KUKA KRL program: wkz1_ab.src, wkz1_ab.dat

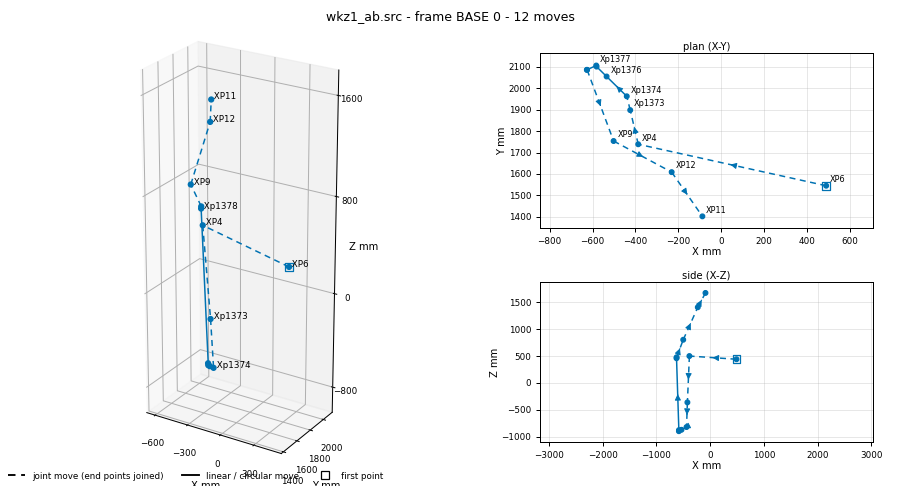
[picture p0: tool path of wkz1_ab.src in frame BASE 0, 12 of 12 moves have a stored position in this frame; points joined in program order, loops and branches not executed]
--- wkz1_ab.src ---
&ACCESS RVP6
&REL 69
&COMMENT Deposita GUN C1
DEF wkz1_ab( )
  ;FOLD INI;%{PE}%V2.2.2,%MKUKATPBASIS,%CINIT,%VCOMMON,%P
  ;FOLD BAS INI;%{PE}%V2.2.2,%MKUKATPBASIS,%CINIT,%VINIT,%P
  INTERRUPT DECL 3 WHEN $STOPMESS==TRUE DO IR_STOPM ( )
  INTERRUPT ON 3
  BAS (#INITMOV,0 )
  ;ENDFOLD
  ;FOLD A20 INI;%{E}%V2.2.2,%MKUKATPA20,%CINIT,%VINIT,%P
  IF ARC20==TRUE THEN
    A20 (ARC_INI)
    INTERRUPT DECL 6 WHEN $CYCFLAG[3]==FALSE DO A20(TECH_STOP2)
  ENDIF
  ;ENDFOLD
  ;FOLD A10 INI;%{E}%V2.2.2,%MKUKATPARC,%CINIT,%VINIT,%P
  IF A10_OPTION==#ACTIVE THEN
    INTERRUPT DECL 4 WHEN $CYCFLAG[2]==FALSE DO A10 (#APPL_ERROR)
    INTERRUPT DECL 7 WHEN A_ARC_SWI==#ACTIVE DO A10 (#ARC_SEAM)
    INTERRUPT DECL 5 WHEN A_FLY_ARC==TRUE DO A10 (#HPU_ARC)
    INTERRUPT  ON 5
    A10_INI ( )
  ENDIF
  ;ENDFOLD
  ;FOLD GRIPPER INI;%{E}%V2.2.2,%MKUKATPGRIPPER,%CINIT,%VINIT,%P
  USER_GRP(0,DUMMY,DUMMY,GDEFAULT)
  ;ENDFOLD
  ;FOLD TOUCHSENSE INI;%{E}%V2.2.2,%MKUKATPTS,%CINIT,%VINIT,%P
  IF H70_OPTION THEN
    INTERRUPT DECL 15 WHEN $MEAS_PULSE[TOUCH_I[TOUCH_ACTIVE].IN_NR] DO H70 (6,CD0 )
    INTERRUPT DECL 16 WHEN $ZERO_MOVE DO H70 (7,CD0 )
    INTERRUPT DECL 17 WHEN $TECHPAR_C[FG_TOUCH,8]>0.5 DO H70 (8,CD0)
    H70 (1,CD0 )
  ENDIF
  ;ENDFOLD
  ;FOLD USER INI;%{P}%V2.2.2,%MKUKATPUSER,%CINIT,%VINIT,%P
  ;Make your modifications here
  ;ENDFOLD
  ;ENDFOLD

; Caracterização dos meios de produção:
; Versão Atual:
; 12/06/2015 12:00 Name: P13.060-R3 CHANGES: Deposita Pinça C1

chk_w1_wechs_ok ( )        ;VERIFICAÇÃO DE FERRAMENTA: c1

;FOLD PTP P6  Vel= 100 % PDAT6 Tool[1]:Gun C1 Base[0];%{PE}%R 4.1.16,%MKUKATPBASIS,%CMOVE,%VPTP,%P 1:PTP, 2:P6, 3:, 5:100, 7:PDAT6
$BWDSTART = FALSE
PDAT_ACT=PPDAT6
BAS(#PTP_DAT)
FDAT_ACT=FP6
BAS(#FRAMES)
BAS(#VEL_PTP,100)
PTP XP6
;ENDFOLD

;FOLD WAIT FOR IN 169 'deposito ocupado'  State= FALSE ;%{PE}%R 4.1.16,%MKUKATPBASIS,%CWAIT_FOR,%VWAIT_FOR,%P 1:0, 2:169, 3:'deposito ocupado', 5:FALSE, 6:
WAIT FOR $IN[169]==FALSE
;ENDFOLD
;FOLD PULSE 175 'protecao da pinca abrir'  State= TRUE   Time= 0.3 sec;%{PE}%R 4.1.16,%MKUKATPBASIS,%COUT,%VPULSE,%P 2:175, 3:'protecao da pinca abrir', 5:TRUE, 6:, 8:0.3
PULSE($OUT[175], TRUE,0.3)
;ENDFOLD
;FOLD WAIT FOR IN 173 'protecao da pinca aberto'  State= TRUE ;%{PE}%R 4.1.16,%MKUKATPBASIS,%CWAIT_FOR,%VWAIT_FOR,%P 1:0, 2:173, 3:'protecao da pinca aberto', 5:TRUE, 6:
WAIT FOR $IN[173]==TRUE
;ENDFOLD
;FOLD WAIT FOR IN 219 'placas de suporte fundidas'  State= TRUE ;%{PE}%R 4.1.16,%MKUKATPBASIS,%CWAIT_FOR,%VWAIT_FOR,%P 1:0, 2:219, 3:'placas de suporte fundidas', 5:TRUE, 6:
WAIT FOR $IN[219]==TRUE
;ENDFOLD
;FOLD WAIT FOR IN 180 'protecao da Garra fechado'  State= TRUE ;%{PE}%R 4.1.16,%MKUKATPBASIS,%CWAIT_FOR,%VWAIT_FOR,%P 1:0, 2:180, 3:'protecao da Garra fechado', 5:TRUE, 6:
WAIT FOR $IN[180]==TRUE
;ENDFOLD

;FOLD PTP P4 CONT Vel= 100 % PDAT4 Tool[1]:Gun C1 Base[0];%{PE}%R 4.1.16,%MKUKATPBASIS,%CMOVE,%VPTP,%P 1:PTP, 2:P4, 3:C_PTP, 5:100, 7:PDAT4
$BWDSTART = FALSE
PDAT_ACT=PPDAT4
BAS(#PTP_DAT)
FDAT_ACT=FP4
BAS(#FRAMES)
BAS(#VEL_PTP,100)
PTP XP4 C_PTP
;ENDFOLD
;FOLD PTP p1373 CONT Vel= 100 % P_OLP2 Tool[1]:Gun C1 Base[0];%{PE}%R 4.1.16,%MKUKATPBASIS,%CMOVE,%VPTP,%P 1:PTP, 2:p1373, 3:C_PTP, 5:100, 7:P_OLP2
$BWDSTART = FALSE
PDAT_ACT=PP_OLP2
BAS(#PTP_DAT)
FDAT_ACT=Fp1373
BAS(#FRAMES)
BAS(#VEL_PTP,100)
PTP Xp1373 C_PTP
;ENDFOLD
;FOLD PTP p1374 CONT Vel= 100 % P_OLP3 Tool[1]:Gun C1 Base[0];%{PE}%R 4.1.16,%MKUKATPBASIS,%CMOVE,%VPTP,%P 1:PTP, 2:p1374, 3:C_PTP, 5:100, 7:P_OLP3
$BWDSTART = FALSE
PDAT_ACT=PP_OLP3
BAS(#PTP_DAT)
FDAT_ACT=Fp1374
BAS(#FRAMES)
BAS(#VEL_PTP,100)
PTP Xp1374 C_PTP
;ENDFOLD
;FOLD LIN p1376  Vel= 0.5 m/s L_OLP1 Tool[1]:Gun C1 Base[0];%{PE}%R 4.1.16,%MKUKATPBASIS,%CMOVE,%VLIN,%P 1:LIN, 2:p1376, 3:, 5:0.5, 7:L_OLP1
$BWDSTART = FALSE
LDAT_ACT=LL_OLP1
BAS(#CP_DAT)
FDAT_ACT=Fp1376
BAS(#FRAMES)
BAS(#VEL_CP,0.5)
LIN Xp1376
;ENDFOLD
;FOLD LIN P10  Vel= 0.5 m/s CPDAT1 Tool[1]:Gun C1 Base[0];%{PE}%R 4.1.16,%MKUKATPBASIS,%CMOVE,%VLIN,%P 1:LIN, 2:P10, 3:, 5:0.5, 7:CPDAT1
$BWDSTART = FALSE
LDAT_ACT=LCPDAT1
BAS(#CP_DAT)
FDAT_ACT=FP10
BAS(#FRAMES)
BAS(#VEL_CP,0.5)
LIN XP10
;ENDFOLD

;FOLD ; Posicao do deposito;%{PE}%R2.2,%MKUKATPBASIS,%CCOMMENT,%VNORMAL,%P 2: Posicao do deposito
;ENDFOLD
;FOLD LIN p1377  Vel= 0.2 m/s CPDAT2 Tool[1]:Gun C1 Base[0];%{PE}%R 4.1.16,%MKUKATPBASIS,%CMOVE,%VLIN,%P 1:LIN, 2:p1377, 3:, 5:0.2, 7:CPDAT2
$BWDSTART = FALSE
LDAT_ACT=LCPDAT2
BAS(#CP_DAT)
FDAT_ACT=Fp1377
BAS(#FRAMES)
BAS(#VEL_CP,0.2)
LIN Xp1377
;ENDFOLD

;FOLD IBUS  OFF;%{PE}%R 4.1.16,%MKUKATPBASIS,%CIBUS,%VMAP,%P 2:#OFF, 3:1
$IBUS_OFF=$IBUS_ON
$IBUS_ON=0
;ENDFOLD
;FOLD WAIT Time= 1 sec;%{PE}%R 4.1.16,%MKUKATPBASIS,%CWAIT,%VWAIT,%P 2:1
WAIT SEC 1
;ENDFOLD
;FOLD WAIT FOR IN 169 'deposito ocupado'  State= TRUE ;%{PE}%R 4.1.16,%MKUKATPBASIS,%CWAIT_FOR,%VWAIT_FOR,%P 1:0, 2:169, 3:'deposito ocupado', 5:TRUE, 6:
WAIT FOR $IN[169]==TRUE
;ENDFOLD
;FOLD OUT 224 'BLOQUEIA MPS'  State= FALSE ;%{PE}%R 4.1.16,%MKUKATPBASIS,%COUT,%VOUTX,%P 2:224, 3:'BLOQUEIA MPS', 5:FALSE, 6:
$OUT[224]=FALSE
;ENDFOLD
;FOLD OUT 223 'Desbloqueio MPS'  State= TRUE ;%{PE}%R 4.1.16,%MKUKATPBASIS,%COUT,%VOUTX,%P 2:223, 3:'Desbloqueio MPS', 5:TRUE, 6:
$OUT[223]=TRUE
;ENDFOLD
;FOLD WAIT FOR IN 217 'MPS destravado'  State= TRUE ;%{PE}%R 4.1.16,%MKUKATPBASIS,%CWAIT_FOR,%VWAIT_FOR,%P 1:0, 2:217, 3:'MPS destravado', 5:TRUE, 6:
WAIT FOR $IN[217]==TRUE
;ENDFOLD
;FOLD WAIT FOR IN 221 'MPS travado'  State= FALSE ;%{PE}%R 4.1.16,%MKUKATPBASIS,%CWAIT_FOR,%VWAIT_FOR,%P 1:0, 2:221, 3:'MPS travado', 5:FALSE, 6:
WAIT FOR $IN[221]==FALSE
;ENDFOLD
;FOLD WAIT Time= 0.5 sec;%{PE}%R 4.1.16,%MKUKATPBASIS,%CWAIT,%VWAIT,%P 2:0.5
WAIT SEC 0.5
;ENDFOLD

;FOLD ; saida sem a pinca;%{PE}%R 4.1.16,%MKUKATPBASIS,%CCOMMENT,%VNORMAL,%P 2:saida sem a pinca
;ENDFOLD
;FOLD LIN p1378 CONT Vel= 0.2 m/s L_OLP3 Tool[8]:Tool Changer Base[0];%{PE}%R 4.1.16,%MKUKATPBASIS,%CMOVE,%VLIN,%P 1:LIN, 2:p1378, 3:C_DIS, 5:0.2, 7:L_OLP3
$BWDSTART = FALSE
LDAT_ACT=LL_OLP3
BAS(#CP_DAT)
FDAT_ACT=Fp1378
BAS(#FRAMES)
BAS(#VEL_CP,0.2)
LIN Xp1378 C_DIS
;ENDFOLD

;FOLD WAIT FOR IN 219 'placas de suporte fundidas'  State= FALSE ;%{PE}%R 4.1.16,%MKUKATPBASIS,%CWAIT_FOR,%VWAIT_FOR,%P 1:0, 2:219, 3:'placas de suporte fundidas', 5:FALSE, 6:
WAIT FOR $IN[219]==FALSE
;ENDFOLD
;FOLD OUT 223 'Desbloqueio MPS'  State= FALSE ;%{PE}%R 4.1.16,%MKUKATPBASIS,%COUT,%VOUTX,%P 2:223, 3:'Desbloqueio MPS', 5:FALSE, 6:
$OUT[223]=FALSE
;ENDFOLD

;FOLD PTP P7 CONT Vel= 100 % PDAT7 Tool[8]:Tool Changer Base[0];%{PE}%R 4.1.16,%MKUKATPBASIS,%CMOVE,%VPTP,%P 1:PTP, 2:P7, 3:C_PTP, 5:100, 7:PDAT7
$BWDSTART = FALSE
PDAT_ACT=PPDAT7
BAS(#PTP_DAT)
FDAT_ACT=FP7
BAS(#FRAMES)
BAS(#VEL_PTP,100)
PTP XP7 C_PTP
;ENDFOLD
;FOLD PTP P9 CONT Vel= 100 % PDAT9 Tool[8]:Tool Changer Base[0];%{PE}%R 4.1.16,%MKUKATPBASIS,%CMOVE,%VPTP,%P 1:PTP, 2:P9, 3:C_PTP, 5:100, 7:PDAT9
$BWDSTART = FALSE
PDAT_ACT=PPDAT9
BAS(#PTP_DAT)
FDAT_ACT=FP9
BAS(#FRAMES)
BAS(#VEL_PTP,100)
PTP XP9 C_PTP
;ENDFOLD
;FOLD PTP P12 CONT Vel= 100 % PDAT11 Tool[8]:Tool Changer Base[0];%{PE}%R 4.1.16,%MKUKATPBASIS,%CMOVE,%VPTP,%P 1:PTP, 2:P12, 3:C_PTP, 5:100, 7:PDAT11
$BWDSTART = FALSE
PDAT_ACT=PPDAT11
BAS(#PTP_DAT)
FDAT_ACT=FP12
BAS(#FRAMES)
BAS(#VEL_PTP,100)
PTP XP12 C_PTP
;ENDFOLD

;FOLD PTP P11  Vel= 100 % PDAT10 Tool[8]:Tool Changer Base[0];%{PE}%R 4.1.16,%MKUKATPBASIS,%CMOVE,%VPTP,%P 1:PTP, 2:P11, 3:, 5:100, 7:PDAT10
$BWDSTART = FALSE
PDAT_ACT=PPDAT10
BAS(#PTP_DAT)
FDAT_ACT=FP11
BAS(#FRAMES)
BAS(#VEL_PTP,100)
PTP XP11
;ENDFOLD

;FOLD PULSE 176 'protecao da pinca fechar'  State= TRUE   Time= 1 sec;%{PE}%R 4.1.16,%MKUKATPBASIS,%COUT,%VPULSE,%P 2:176, 3:'protecao da pinca fechar', 5:TRUE, 6:, 8:1
PULSE($OUT[176], TRUE,1)
;ENDFOLD

END

--- wkz1_ab.dat ---
&ACCESS RVP6
&REL 69
&COMMENT Deposita GUN C1
DEFDAT  WKZ1_AB
;FOLD EXTERNAL DECLARATIONS;%{PE}%V2.2.2,%MKUKATPBASIS,%CEXT,%VCOMMON,%P
;FOLD BAS EXT;%{PE}%V2.2.2,%MKUKATPBASIS,%CEXT,%VEXT,%P
EXT  BAS (BAS_COMMAND  :IN,REAL  :IN )
DECL INT SUCCESS
;ENDFOLD
;FOLD A10 EXT;%{E}%V2.2.2,%MKUKATPARC,%CEXT,%VEXT,%P
EXT  A10 (A_CMD_T  :IN,A_STRT_T  :IN,A_WELD_T  :IN,A_END_T  :IN,INT  :IN )
;ENDFOLD
;FOLD A20 EXT;%{E}%V2.2.2,%MKUKATPA20,%CEXT,%VEXT,%P
EXT  A20 (INT  :IN,WELD_ST  :IN,WELD_FI  :IN,INT  :IN )
;ENDFOLD
;FOLD GRIPPER EXT;%{E}%V2.2.2,%MKUKATPGRIPPER,%CEXT,%VEXT,%P
EXT  H50 (INT  :IN,INT  :IN,INT  :IN,GRP_TYP  :IN )
;ENDFOLD
;FOLD SPOT EXT;%{E}%V2.2.2,%MKUKATPSPOT,%CEXT,%VEXT,%P
EXT  USERSPOT (S_COMMAND  :IN,SPOT_TYPE  :IN )
;ENDFOLD
;FOLD TOUCHSENSE EXT;%{E}%V2.2.2,%MKUKATPTS,%CEXT,%VEXT,%P
EXT  H70 (INT  :IN,SRCH_TYP_2  :OUT,E6POS  :IN,SRCH_TYP_3  :IN,SRCH_TYP_2  :IN,SRCH_TYP_2  :IN,SRCH_TYP_2  :IN,SRCH_TYP_2  :IN,SRCH_TYP_2  :IN,INT  :IN )
;ENDFOLD
;FOLD USER EXT;%{}%V2.2.2,%MKUKATPUSER,%CEXT,%VEXT,%P
;Make here your modifications
;ENDFOLD
;ENDFOLD

;# ============ START PATH : za_p13060r3_c1 =============
DECL FDAT Fp1373={TOOL_NO 1,BASE_NO 0,IPO_FRAME #BASE}
DECL PDAT PP_OLP2={VEL 100.0,ACC 100.0,APO_DIST 20.0}
DECL E6POS Xp1373={x -424.213287,y 1897.96704,z -363.086609,a 25.8961792,b 0.644996405,c 3.42784691,s 2,t 11,e1 0.0,e2 0.0,e3 0.0,e4 0.0,e5 0.0,e6 0.0}
DECL FDAT Fp1374={TOOL_NO 1,BASE_NO 0,IPO_FRAME #BASE}
DECL PDAT PP_OLP3={VEL 100.0,ACC 100.0,APO_DIST 10.0}
DECL E6POS Xp1374={x -440.401489,y 1962.54797,z -822.446411,a 15.2994604,b 0.811248183,c 0.186222494,s 2,t 11,e1 0.0,e2 0.0,e3 0.0,e4 0.0,e5 0.0,e6 0.0}
DECL FDAT Fp1376={TOOL_NO 1,BASE_NO 0,IPO_FRAME #BASE}
DECL E6POS Xp1376={x -534.518005,y 2054.86011,z -873.282776,a 15.3016195,b 0.811761796,c 0.184798405,s 2,t 11,e1 0.0,e2 0.0,e3 0.0,e4 0.0,e5 0.0,e6 0.0}
DECL LDAT LL_OLP1={VEL 0.5,ACC 100.0,APO_DIST 1.0,APO_FAC 100.0}
DECL FDAT Fp1377={TOOL_NO 1,BASE_NO 0,IPO_FRAME #BASE}
DECL E6POS Xp1377={x -582.689392,y 2106.07202,z -899.922913,a 15.2830095,b 0.816190898,c 0.34551689,s 2,t 11,e1 0.0,e2 0.0,e3 0.0,e4 0.0,e5 0.0,e6 0.0}
DECL FDAT Fp1378={TOOL_NO 8,BASE_NO 0,IPO_FRAME #BASE}
DECL E6POS Xp1378={x -626.691589,y 2086.03101,z 458.803711,a -44.7220497,b 0.70728451,c 179.466003,s 2,t 11,e1 0.0,e2 0.0,e3 0.0,e4 0.0,e5 0.0,e6 0.0}
DECL LDAT LL_OLP3={VEL 0.5,ACC 85.0,APO_DIST 2.0,APO_FAC 0.0}
DECL BASIS_SUGG_T LAST_BASIS={POINT1[] "P12                     ",POINT2[] "P12                     ",CP_PARAMS[] "CPDAT1                  ",PTP_PARAMS[] "PDAT11                  ",CONT[] "                        ",CP_VEL[] "0.2                     ",PTP_VEL[] "80                      "}
DECL E6POS XP4={x -386.9086,y 1738.698,z 500.014313,a 28.7212296,b -2.10732794,c 14.1292801,s 2,t 11,e1 0.0,e2 0.0,e3 0.0,e4 0.0,e5 0.0,e6 0.0}
DECL FDAT FP4={TOOL_NO 1,BASE_NO 0,IPO_FRAME #BASE}
DECL PDAT PPDAT4={VEL 100.0,ACC 100.0,APO_DIST 50.0}
DECL E6POS XP6={x 489.958496,y 1545.21301,z 440.531189,a 63.9639511,b -7.4234581,c 1.31531894,s 2,t 11,e1 0.0,e2 0.0,e3 0.0,e4 0.0,e5 0.0,e6 0.0}
DECL FDAT FP6={TOOL_NO 1,BASE_NO 0,IPO_FRAME #BASE}
DECL PDAT PPDAT6={VEL 100.0,ACC 100.0,APO_DIST 10.0}
DECL E6POS XP7={x -625.279419,y 2085.8291,z 477.282013,a -44.7222404,b 0.708276987,c 179.466202,s 2,t 11,e1 0.0,e2 0.0,e3 0.0,e4 0.0,e5 0.0,e6 0.0}
DECL FDAT FP7={TOOL_NO 8,BASE_NO 0,IPO_FRAME #BASE}
DECL PDAT PPDAT7={VEL 100.0,ACC 100.0,APO_DIST 10.0}
DECL E6POS XP9={x -501.769714,y 1753.83997,z 803.569275,a -44.7246284,b 3.61455107,c 179.398102,s 2,t 11,e1 0.0,e2 0.0,e3 0.0,e4 0.0,e5 0.0,e6 0.0}
DECL FDAT FP9={TOOL_NO 8,BASE_NO 0,IPO_FRAME #BASE}
DECL PDAT PPDAT9={VEL 100.0,ACC 100.0,APO_DIST 50.0}
DECL E6POS XP10={x -581.368408,y 2101.01001,z -879.867615,a 15.2993603,b 0.811329722,c 0.178669199,s 2,t 11,e1 0.0,e2 0.0,e3 0.0,e4 0.0,e5 0.0,e6 0.0}
DECL FDAT FP10={TOOL_NO 1,BASE_NO 0,IPO_FRAME #BASE}
DECL LDAT LCPDAT1={VEL 2.0,ACC 100.0,APO_DIST 100.0,APO_FAC 50.0}
DECL LDAT LCPDAT2={VEL 2.0,ACC 90.0,APO_DIST 100.0,APO_FAC 50.0}
DECL E6POS XP11={x -87.5717773,y 1402.37598,z 1675.646,a -69.6122437,b 42.7373886,c -162.170502,s 2,t 3,e1 0.0,e2 0.0,e3 0.0,e4 0.0,e5 0.0,e6 0.0}
DECL FDAT FP11={TOOL_NO 8,BASE_NO 0,IPO_FRAME #BASE}
DECL PDAT PPDAT10={VEL 100.0,ACC 100.0,APO_DIST 10.0}
DECL E6POS XP12={x -230.829498,y 1608.68896,z 1409.09998,a -61.1877708,b 27.0093708,c -166.5439,s 2,t 3,e1 0.0,e2 0.0,e3 0.0,e4 0.0,e5 0.0,e6 0.0}
DECL FDAT FP12={TOOL_NO 8,BASE_NO 0,IPO_FRAME #BASE}
DECL PDAT PPDAT11={VEL 100.0,ACC 100.0,APO_DIST 100.0}
ENDDAT
